{attribute addProperty BoxType "EL2521--0000"}
{attribute addProperty Id "InputsAT %I*Inputs_406D1DC23240OutputsAT %Q*Outputs_5374A1F83240WcStateAT %I*WcState_98A4DF7520.250InfoDataAT %I*InfoData_BC63D37F80100"}
{attribute addProperty CRC "4124668444"}
{attribute addProperty SizeInBites "146"}
{attribute addProperty SizeInBytes "18.25"}
TYPE EL2521_7A3DFE70 :
STRUCT
	{attribute addProperty Name "Inputs"}
	Inputs : Inputs_406D1DC2;
	{attribute addProperty Name "Outputs"}
	Outputs : Outputs_5374A1F8;
	{attribute addProperty Name "WcState"}
	WcState : WcState_98A4DF75;
	{attribute addProperty Name "InfoData"}
	InfoData : InfoData_BC63D37F;
END_STRUCT
END_TYPE

(* stored: Version 1.2.0.0, ProductVersion 3.1.4024.9
   DUT EL2521_7A3DFE70: Id {df2b9b84-9bc5-473d-87da-863e650f4e91} *)
